{attribute 'linkalways'} 
{attribute 'no_explicit_call' := 'This FB is a CLASS and must be accessed using methods or properties'}
{attribute 'enable_dynamic_creation'}
FUNCTION_BLOCK PUBLIC PreExecutionCheckFailedAlarm EXTENDS Alarm
VAR
	state : (CLEARED, RAISED);
	_reason : T_MAXSTRING;
END_VAR

PROPERTY Active : BOOL
GET
Active := state <> CLEARED;
END_GET
END_PROPERTY

METHOD PUBLIC Clear
_reason := '';
state := CLEARED;
END_METHOD

PROPERTY PUBLIC Message : T_MaxString
GET
Message := 'Pre-execution check failed';
END_GET
END_PROPERTY

METHOD PUBLIC Raise
VAR_INPUT
	Reason : T_MAXSTRING;
END_VAR
_reason := Reason;
state := RAISED;
END_METHOD

PROPERTY Reason : T_MaxString
GET
Reason := _reason;
END_GET
END_PROPERTY

END_FUNCTION_BLOCK

(* stored: Version 1.1.0.1, ProductVersion 3.1.4024.13
   POU PreExecutionCheckFailedAlarm: Id {19838939-01da-0cdc-0757-d5a321df90da}, SpecialFunc None
   Property Active: Id {b461f2e3-1093-01b1-37b4-2c664a29ac7c}
   Get Get: Id {6780eeae-e68c-03f8-10b9-0fabe8985792}
   Method Clear: Id {ca9e6e1e-d3c6-0ea1-21de-a7876ed5f8b6}
   Property Message: Id {e6e11f9d-2d9e-011b-3665-ca6a5ddf0c42}
   Get Get: Id {0dfe35ee-1ad1-0be3-182f-6120a1cb4f77}
   Method Raise: Id {c5478646-dc30-0190-2385-8e664552a648}
   Property Reason: Id {7d4a7d11-9473-03d1-210b-0d8f8f567841}
   Get Get: Id {3e1ad541-038e-0c24-0e43-c70e5ca018c6} *)
